Universal Robots PolyScope program: gravityFeederZ.urp

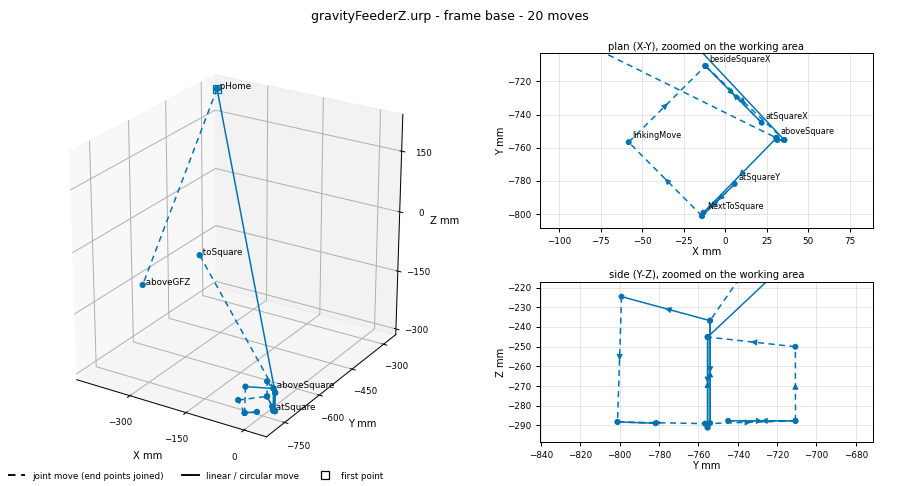
[picture p0: tool path of gravityFeederZ.urp in frame base, 20 of 23 moves have a stored position in this frame; points joined in program order, loops and branches not executed]
Program gravityFeederZ (installation=admin directory=/programs/WED_9AM createdIn=3.8.0.61336 lastSavedIn=3.15.8.106339 robotSerialNumber=2015350925)
Calibrated DH parameters: a=[0.000202, -0.047961, -0.392055, -0.000001, 0.000007, 0]; d=[0.089082, 828.736652, -823.627268, -4.999465, 0.094767, 0.082274]; alpha=[1.570325, 0.00051, -0.003464, 1.570175, -1.569769, 0]; deltaTheta=[0.000028, 1.457808, -1.502844, -6.238105, -6.283148, -0.000082]
Robot Program (runOnlyOnce=true)
  Set DigitalOutput pin=digital_out[0]; digitalValue=0
  Call _adminLinearIndex3
  MoveJ speed 180 deg/s, acceleration 100 deg/s^2 (useActiveTCP=true)
    Waypoint pHome: TCP in base x=-424.566 y=-265.032 z=215.658 mm, rx=-1.1995 ry=-2.8938 rz=-0.0046 rad; joints [224.997, -90.003, -90.003, -90.012, 89.253, -0.016] deg; flange x=-423.002 y=-266.37 z=431.548 mm, rx=-1.1995 ry=-2.8938 rz=-0.0046 rad
    Waypoint aboveGFZ: TCP in base x=-332.198 y=-721.027 z=-91.342 mm, rx=-1.1458 ry=-2.7483 rz=0.4618 rad; joints [257.098, -133.024, -83.899, -36.825, 79.777, 30.704] deg; flange x=-281.911 y=-671.438 z=112.68 mm, rx=-1.1458 ry=-2.7483 rz=0.4618 rad
  MoveL speed 250 mm/s, acceleration 1200 mm/s^2 (useActiveTCP=true) feature=GravityFeeder
    Waypoint atGFRel (Relative): relativeFromPosition TCP in base x=-332.161 y=-721.02 z=-91.333 mm, rx=-1.1456 ry=-2.7483 rz=0.4618 rad; joints [257.1, -133.021, -83.905, -36.821, 79.779, 30.701] deg; TCP in base x=-349.623 y=-738.215 z=-134.704 mm, rx=-1.1458 ry=-2.7483 rz=0.4617 rad; joints [256.049, -139.138, -79.818, -34.619, 80.085, 29.68] deg; pose in feature x=383.721 y=-143.056 z=-429.589 mm, rx=0.0049 ry=-3.1277 rz=-0.0208 rad; flange x=-299.348 y=-688.635 z=69.324 mm, rx=-1.1458 ry=-2.7483 rz=0.4617 rad
    Set DigitalOutput pin=digital_out[0]; digitalValue=1
    Wait Sleep waitTime=1
    Waypoint moveUpRel (Relative): motionParameters(jointSpeed=1.047198 jointAcceleration=1.396263 cartesianSpeed=0.08 cartesianAcceleration=0.08); relativeFromPosition TCP in base x=-349.679 y=-738.175 z=-134.732 mm, rx=-1.1458 ry=-2.7482 rz=0.4615 rad; joints [256.047, -139.14, -79.817, -34.622, 80.078, 29.678] deg; TCP in base x=-352.177 y=-740.693 z=-133.441 mm, rx=-1.1459 ry=-2.7483 rz=0.4616 rad; joints [255.899, -139.389, -79.072, -35.092, 80.127, 29.538] deg; pose in feature x=383.695 y=-146.833 z=-429.609 mm, rx=0.0048 ry=-3.1277 rz=-0.0208 rad; flange x=-301.909 y=-691.121 z=70.59 mm, rx=-1.1459 ry=-2.7483 rz=0.4616 rad
    Waypoint aboveGFRel (Relative): relativeFromPosition TCP in base x=-352.168 y=-740.682 z=-133.466 mm, rx=-1.1459 ry=-2.7483 rz=0.4615 rad; joints [255.9, -139.39, -79.072, -35.094, 80.127, 29.537] deg; TCP in base x=-335.923 y=-723.364 z=-67.573 mm, rx=-1.1459 ry=-2.7483 rz=0.4618 rad; joints [256.839, -131.557, -82.429, -39.719, 79.848, 30.464] deg; pose in feature x=383.739 y=-146.867 z=-359.588 mm, rx=0.0048 ry=-3.1278 rz=-0.0207 rad; flange x=-285.658 y=-673.766 z=136.452 mm, rx=-1.1459 ry=-2.7483 rz=0.4618 rad
  MoveJ speed 60 deg/s, acceleration 80 deg/s^2 (useActiveTCP=true)
    Waypoint toSquare: TCP in base x=-247.912 y=-616.312 z=-38.501 mm, rx=-1.0104 ry=-2.8148 rz=0.3601 rad; joints [262.227, -115.472, -102.903, -39.652, 79.845, 30.465] deg; flange x=-204.646 y=-577.614 z=169.45 mm, rx=-1.0104 ry=-2.8148 rz=0.3601 rad
    Waypoint aboveSquare: TCP in base x=30.853 y=-754.073 z=-236.789 mm, rx=1.2016 ry=2.8995 rz=-0.0036 rad; joints [280.731, -146.973, -74.414, -48.471, 89.941, 55.557] deg; flange x=30.445 y=-753.369 z=-20.89 mm, rx=1.2016 ry=2.8995 rz=-0.0036 rad
  MoveL speed 250 mm/s, acceleration 1200 mm/s^2 (useActiveTCP=true) feature=Base
    Waypoint atSquare: TCP in base x=30.839 y=-754.011 z=-288.826 mm, rx=1.2017 ry=2.8994 rz=-0.0033 rad; joints [280.732, -151.989, -73.416, -44.462, 89.958, 55.554] deg; flange x=30.419 y=-753.34 z=-72.928 mm, rx=1.2017 ry=2.8994 rz=-0.0033 rad
    Set DigitalOutput pin=digital_out[0]; digitalValue=0
    Wait Sleep waitTime=1
    Waypoint aboveSquare: TCP in base x=30.853 y=-754.073 z=-236.789 mm, rx=1.2016 ry=2.8995 rz=-0.0036 rad; joints [280.731, -146.973, -74.414, -48.471, 89.941, 55.557] deg; flange x=30.445 y=-753.369 z=-20.89 mm, rx=1.2016 ry=2.8995 rz=-0.0036 rad
    Waypoint NextToSquare: TCP in base x=-13.128 y=-799.041 z=-224.591 mm, rx=1.2019 ry=2.8993 rz=-0.0035 rad; joints [276.969, -151.009, -63.364, -55.49, 89.947, 51.825] deg; flange x=-13.559 y=-798.339 z=-8.693 mm, rx=1.2019 ry=2.8993 rz=-0.0035 rad
    Set DigitalOutput pin=digital_out[0]; digitalValue=1
  MoveJ speed 180 deg/s, acceleration 100 deg/s^2 (useActiveTCP=true)
    Waypoint besideSquareY: TCP in base x=-13.979 y=-801.074 z=-288.268 mm, rx=1.2017 ry=2.8993 rz=-0.0034 rad; joints [276.893, -157.027, -61.628, -51.212, 89.962, 51.732] deg; flange x=-14.421 y=-800.39 z=-72.369 mm, rx=1.2017 ry=2.8993 rz=-0.0034 rad
  Wait Sleep waitTime=0.1
  MoveL speed 30 mm/s, acceleration 30 mm/s^2 (useActiveTCP=true) feature=Base
    If force()≤45 (checkContinuously=true)
      Waypoint atSquareY: TCP in base x=5.704 y=-781.743 z=-288.921 mm, rx=1.2018 ry=2.8994 rz=-0.0034 rad; joints [278.513, -154.846, -66.757, -48.267, 89.956, 53.347] deg; flange x=5.291 y=-781.072 z=-73.022 mm, rx=1.2018 ry=2.8994 rz=-0.0034 rad
    Wait Sleep waitTime=0.5
  MoveJ speed 180 deg/s, acceleration 100 deg/s^2 (useActiveTCP=true)
    Waypoint besideSquareY: TCP in base x=-13.979 y=-801.074 z=-288.268 mm, rx=1.2017 ry=2.8993 rz=-0.0034 rad; joints [276.893, -157.027, -61.628, -51.212, 89.962, 51.732] deg; flange x=-14.421 y=-800.39 z=-72.369 mm, rx=1.2017 ry=2.8993 rz=-0.0034 rad
    Waypoint linkingMove: motionParameters(blendRadius=0.005); TCP in base x=-58.166 y=-756.622 z=-289.108 mm, rx=1.2018 ry=2.8995 rz=-0.0034 rad; joints [273.941, -152.445, -72.394, -45.037, 89.973, 48.766] deg; flange x=-58.56 y=-755.949 z=-73.21 mm, rx=1.2018 ry=2.8995 rz=-0.0034 rad
    Waypoint besideSquareX: TCP in base x=-11.935 y=-710.663 z=-287.721 mm, rx=1.2018 ry=2.8995 rz=-0.0031 rad; joints [277.945, -147.814, -83.221, -38.844, 89.981, 52.757] deg; flange x=-12.351 y=-710.027 z=-71.823 mm, rx=1.2018 ry=2.8995 rz=-0.0031 rad
  Wait Sleep waitTime=0.1
  MoveL speed 30 mm/s, acceleration 30 mm/s^2 (useActiveTCP=true) feature=Base
    If force()≤45 (checkContinuously=true)
      Waypoint atSquareX: TCP in base x=21.933 y=-744.88 z=-287.695 mm, rx=1.2021 ry=2.8994 rz=-0.0034 rad; joints [280.186, -150.95, -75.639, -43.281, 89.954, 55.017] deg; flange x=21.547 y=-744.217 z=-71.796 mm, rx=1.2021 ry=2.8994 rz=-0.0034 rad
    Wait Sleep waitTime=0.5
  MoveJ speed 60 deg/s, acceleration 80 deg/s^2 (useActiveTCP=true)
    Waypoint besideSquareX: motionParameters(jointSpeed=1.047198 jointAcceleration=1.047198 cartesianSpeed=0.25 cartesianAcceleration=1.2); TCP in base x=-11.935 y=-710.663 z=-287.721 mm, rx=1.2018 ry=2.8995 rz=-0.0031 rad; joints [277.945, -147.814, -83.221, -38.844, 89.981, 52.757] deg; flange x=-12.351 y=-710.027 z=-71.823 mm, rx=1.2018 ry=2.8995 rz=-0.0031 rad
    Waypoint linkingMove2: TCP in base x=-11.939 y=-710.712 z=-250.057 mm, rx=1.2018 ry=2.8994 rz=-0.0033 rad; joints [277.941, -143.93, -84.001, -41.939, 89.971, 52.763] deg; flange x=-12.359 y=-710.042 z=-34.158 mm, rx=1.2018 ry=2.8994 rz=-0.0033 rad
    Waypoint aboveSquare2: TCP in base x=35.572 y=-755.293 z=-245.106 mm, rx=1.2015 ry=2.8995 rz=-0.0035 rad; joints [281.069, -147.899, -73.981, -47.981, 89.941, 55.891] deg; flange x=35.168 y=-754.6 z=-29.207 mm, rx=1.2015 ry=2.8995 rz=-0.0035 rad
    Set DigitalOutput pin=digital_out[0]; digitalValue=0
    Wait Sleep waitTime=1
  MoveL speed 250 mm/s, acceleration 1200 mm/s^2 (useActiveTCP=true) feature=Base
    Waypoint atSquare2: TCP in base x=35.521 y=-755.31 z=-291.084 mm, rx=1.2016 ry=2.8995 rz=-0.0035 rad; joints [281.068, -152.362, -73.004, -44.493, 89.953, 55.883] deg; flange x=35.113 y=-754.613 z=-75.186 mm, rx=1.2016 ry=2.8995 rz=-0.0035 rad
    Set DigitalOutput pin=digital_out[0]; digitalValue=1
    Wait Sleep waitTime=1
    Waypoint easeOut: TCP in base x=31.269 y=-755.318 z=-291.081 mm, rx=1.2017 ry=2.8995 rz=-0.0035 rad; joints [280.748, -152.344, -73.045, -44.471, 89.952, 55.567] deg; flange x=30.868 y=-754.623 z=-75.183 mm, rx=1.2017 ry=2.8995 rz=-0.0035 rad
    Waypoint aboveSquare2: TCP in base x=35.572 y=-755.293 z=-245.106 mm, rx=1.2015 ry=2.8995 rz=-0.0035 rad; joints [281.069, -147.899, -73.981, -47.981, 89.941, 55.891] deg; flange x=35.168 y=-754.6 z=-29.207 mm, rx=1.2015 ry=2.8995 rz=-0.0035 rad
  MoveL speed 250 mm/s, acceleration 1200 mm/s^2 (useActiveTCP=true) feature=Base
    Waypoint pHome: TCP in base x=-424.566 y=-265.032 z=215.658 mm, rx=-1.1995 ry=-2.8938 rz=-0.0046 rad; joints [224.997, -90.003, -90.003, -90.012, 89.253, -0.016] deg; flange x=-423.002 y=-266.37 z=431.548 mm, rx=-1.1995 ry=-2.8938 rz=-0.0046 rad
SubProgram -> _adminLinearIndex3
SubProgram _adminLinearIndex3 (keepSynchronizedWithDisk=false) programFile=/programs/me345_admin/_adminLinearIndex3.urp
  Folder Move_linear_slide_Index3
    var_1 := False
    Loop While (checkContinuously=false) expression=var_1≟ False
      var_1 := socket_open("10.241.34.48",4001)
    var_3 := 1
    Send := "s r0x24 21"
    Script: socket_send_string(Send)
    Script: socket_send_byte(13)
    Send_Reply := socket_read_string()
    Send := "s r0xca 112778"
    Script: socket_send_string(Send)
    Script: socket_send_byte(13)
    Send_Reply := socket_read_string()
    Send := "t 1"
    Script: socket_send_string(Send)
    Script: socket_send_byte(13)
    Send_Reply := socket_read_string()
    Loop While (checkContinuously=false) expression=var_3≠0
      Send := "g r0xA0"
      Script: socket_send_string(Send)
      Script: socket_send_byte(13)
      var_3 := socket_get_var("v")
      Wait Sleep waitTime=0.1
    Script: socket_close()
    Script: sync()
